Fanuc KAREL source: ko00014.KL

-- PROVISIONAL review KL for V770-1; original PC SHA256 38a8e8a560263ba2283a1afa9c0beebb30bd2b0d958a9f8d6977a9dd7e8083db
-- Incomplete behavior may be omitted. Consult companion uncertainty JSON. Do not deploy.
PROGRAM KO00014
%NOLOCKGROUP
-- UNRESOLVED_DECL P1 type=000102
-- UNRESOLVED_DECL P2 type=000102
-- UNRESOLVED_DECL P3 type=000102
-- UNRESOLVED_DECL P4 type=000102
-- UNRESOLVED_DECL OUT type=000102
BEGIN
  -- UNRESOLVED_PC offsets 5-80; opcodes 27,27,49,7E,AD,27,49,7E,AD,27,49,7E,AD,27,49,7E,AD,76,7E,4A
  -- UNRESOLVED_PC offsets 85-89; opcodes 7F
END KO00014
